_CFC_ (* Continuous Function Chart, elements in execution order *)
(* 60s *)
#0 AND(#2.Xm, SHU6_P2_UST_RE_RABOTA)
#1 ADD(SHU6_P2_M_MINSPEED, 0.1)
#2 LT_HZm20:ISTOK_LT(dost: TRUE, x: SHU6_P2_SPEEDMOTOR, ust: #1, shkal: -, gist: 1)
#3 INT_TO_TIME(SHU6_P2_M_ZAD_HZM20)
#4 MUL(#3, 1000)
#5 TON_HZm20:TON(IN: #0, PT: #4)
#6 AND(#5.Q, NOT SHU6_P2_M_SB2_STER_REG)
#7 SR_HZ20S60:SR(SET1: #6, RESET: SHU6_P2_SB)
#8 SHU6_P2_HZ20S60 <= #7.Q1
_END_CFC_
(* the same logic as Structured Text *)
(* 60s *)
_t19 := LT_HZm20.Xm AND SHU6_P2_UST_RE_RABOTA;
LT_HZm20(dost := TRUE, x := SHU6_P2_SPEEDMOTOR, ust := SHU6_P2_M_MINSPEED + 0.1, gist := 1);
TON_HZm20(IN := _t19, PT := INT_TO_TIME(SHU6_P2_M_ZAD_HZM20) * 1000);
SR_HZ20S60(SET1 := TON_HZm20.Q AND NOT SHU6_P2_M_SB2_STER_REG, RESET := SHU6_P2_SB);
SHU6_P2_HZ20S60 := SR_HZ20S60.Q1;
END_PROGRAM

(* POU TZBiS/TZB/Z_ALL, CFC *)
PROGRAM Z_ALL
VAR
	SR_Z_all: SR;
END_VAR
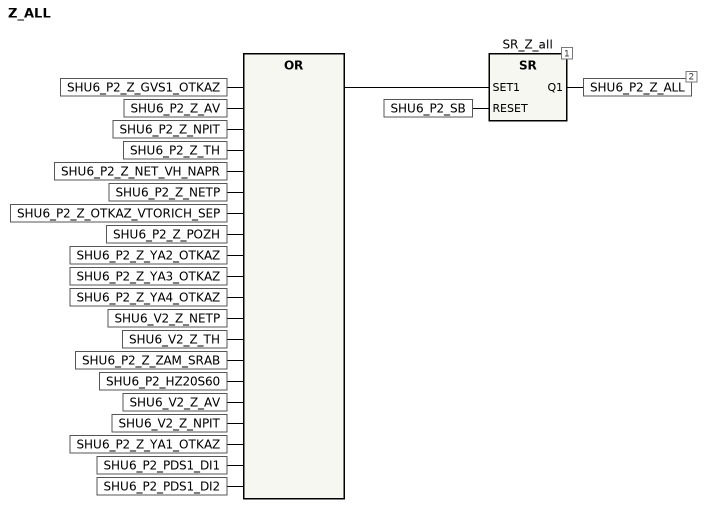
_CFC_ (* Continuous Function Chart, elements in execution order *)
#0 OR(SHU6_P2_Z_GVS1_OTKAZ, SHU6_P2_Z_AV, SHU6_P2_Z_NPIT, SHU6_P2_Z_TH, SHU6_P2_Z_NET_VH_NAPR, SHU6_P2_Z_NETP, SHU6_P2_Z_OTKAZ_VTORICH_SEP, SHU6_P2_Z_POZH, SHU6_P2_Z_YA2_OTKAZ, SHU6_P2_Z_YA3_OTKAZ, SHU6_P2_Z_YA4_OTKAZ, SHU6_V2_Z_NETP, SHU6_V2_Z_TH, SHU6_P2_Z_ZAM_SRAB, SHU6_P2_HZ20S60, SHU6_V2_Z_AV, SHU6_V2_Z_NPIT, SHU6_P2_Z_YA1_OTKAZ, SHU6_P2_PDS1_DI1, SHU6_P2_PDS1_DI2)
#1 SR_Z_all:SR(SET1: #0, RESET: SHU6_P2_SB)
#2 SHU6_P2_Z_ALL <= #1.Q1
_END_CFC_
(* the same logic as Structured Text *)
SR_Z_all(SET1 := SHU6_P2_Z_GVS1_OTKAZ OR SHU6_P2_Z_AV OR SHU6_P2_Z_NPIT OR SHU6_P2_Z_TH OR SHU6_P2_Z_NET_VH_NAPR OR SHU6_P2_Z_NETP OR SHU6_P2_Z_OTKAZ_VTORICH_SEP OR SHU6_P2_Z_POZH OR SHU6_P2_Z_YA2_OTKAZ OR SHU6_P2_Z_YA3_OTKAZ OR SHU6_P2_Z_YA4_OTKAZ OR SHU6_V2_Z_NETP OR SHU6_V2_Z_TH OR SHU6_P2_Z_ZAM_SRAB OR SHU6_P2_HZ20S60 OR SHU6_V2_Z_AV OR SHU6_V2_Z_NPIT OR SHU6_P2_Z_YA1_OTKAZ OR SHU6_P2_PDS1_DI1 OR SHU6_P2_PDS1_DI2, RESET := SHU6_P2_SB);
SHU6_P2_Z_ALL := SR_Z_all.Q1;
END_PROGRAM

(* POU TZBiS/TZB/Z_YA2_Otk, CFC *)
PROGRAM Z_YA2_Otk
VAR
	SR_YA2_Otkaz: SR;
	TON_YA2_Otk: TON;
	TON_YA2_N_OTKR: TON;
	TON_YA2_N_ZAKR: TON;
	TON_YA2_ZKR: TON;
	TON_AVT: TON;

	a: BOOL;
	b: BOOL;
	c: BOOL;
	d: BOOL;
	e: BOOL;
END_VAR
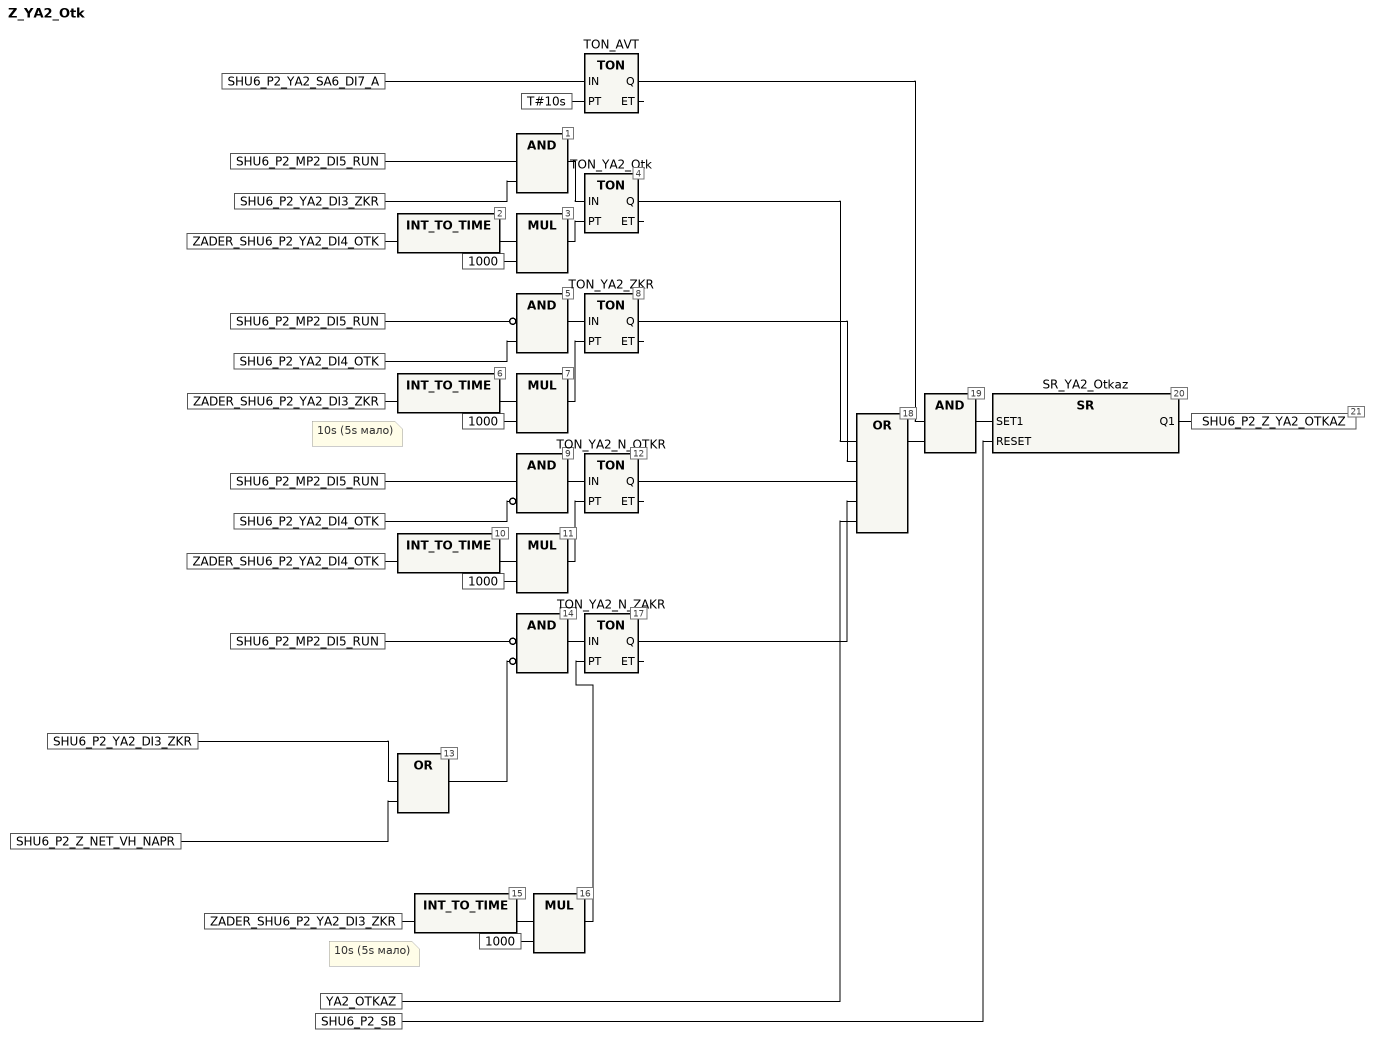
_CFC_ (* Continuous Function Chart, elements in execution order *)
(* 10s (5s мало) *)
(* 10s (5s мало) *)
#0 TON_AVT:TON(IN: SHU6_P2_YA2_SA6_DI7_A, PT: T#10s)
#1 AND(SHU6_P2_MP2_DI5_RUN, SHU6_P2_YA2_DI3_ZKR)
#2 INT_TO_TIME(ZADER_SHU6_P2_YA2_DI4_OTK)
#3 MUL(#2, 1000)
#4 TON_YA2_Otk:TON(IN: #1, PT: #3)
#5 AND(NOT SHU6_P2_MP2_DI5_RUN, SHU6_P2_YA2_DI4_OTK)
#6 INT_TO_TIME(ZADER_SHU6_P2_YA2_DI3_ZKR)
#7 MUL(#6, 1000)
#8 TON_YA2_ZKR:TON(IN: #5, PT: #7)
#9 AND(SHU6_P2_MP2_DI5_RUN, NOT SHU6_P2_YA2_DI4_OTK)
#10 INT_TO_TIME(ZADER_SHU6_P2_YA2_DI4_OTK)
#11 MUL(#10, 1000)
#12 TON_YA2_N_OTKR:TON(IN: #9, PT: #11)
#13 OR(SHU6_P2_YA2_DI3_ZKR, SHU6_P2_Z_NET_VH_NAPR)
#14 AND(NOT SHU6_P2_MP2_DI5_RUN, NOT #13)
#15 INT_TO_TIME(ZADER_SHU6_P2_YA2_DI3_ZKR)
#16 MUL(#15, 1000)
#17 TON_YA2_N_ZAKR:TON(IN: #14, PT: #16)
#18 OR(#4.Q, #8.Q, #12.Q, #17.Q, YA2_OTKAZ)
#19 AND(#0.Q, #18)
#20 SR_YA2_Otkaz:SR(SET1: #19, RESET: SHU6_P2_SB)
#21 SHU6_P2_Z_YA2_OTKAZ <= #20.Q1
_END_CFC_
(* the same logic as Structured Text *)
(* 10s (5s мало) *)
(* 10s (5s мало) *)
TON_AVT(IN := SHU6_P2_YA2_SA6_DI7_A, PT := T#10s);
TON_YA2_Otk(IN := SHU6_P2_MP2_DI5_RUN AND SHU6_P2_YA2_DI3_ZKR, PT := INT_TO_TIME(ZADER_SHU6_P2_YA2_DI4_OTK) * 1000);
TON_YA2_ZKR(IN := NOT SHU6_P2_MP2_DI5_RUN AND SHU6_P2_YA2_DI4_OTK, PT := INT_TO_TIME(ZADER_SHU6_P2_YA2_DI3_ZKR) * 1000);
TON_YA2_N_OTKR(IN := SHU6_P2_MP2_DI5_RUN AND NOT SHU6_P2_YA2_DI4_OTK, PT := INT_TO_TIME(ZADER_SHU6_P2_YA2_DI4_OTK) * 1000);
TON_YA2_N_ZAKR(IN := NOT SHU6_P2_MP2_DI5_RUN AND NOT (SHU6_P2_YA2_DI3_ZKR OR SHU6_P2_Z_NET_VH_NAPR), PT := INT_TO_TIME(ZADER_SHU6_P2_YA2_DI3_ZKR) * 1000);
SR_YA2_Otkaz(SET1 := TON_AVT.Q AND (TON_YA2_Otk.Q OR TON_YA2_ZKR.Q OR TON_YA2_N_OTKR.Q OR TON_YA2_N_ZAKR.Q OR YA2_OTKAZ), RESET := SHU6_P2_SB);
SHU6_P2_Z_YA2_OTKAZ := SR_YA2_Otkaz.Q1;
END_PROGRAM

(* POU TZBiS/TZB/Z_YA1_YA2_NPit, CFC *)
PROGRAM Z_YA1_YA2_NPit
VAR
	SR_YA1_YA2_NPit: SR;
	SR_IBP_NPit: SR;
	SR_A1_G1_NPit: SR;
	SR_A1_TV1_NPit: SR;
	SR_24V_NPit: SR;
END_VAR
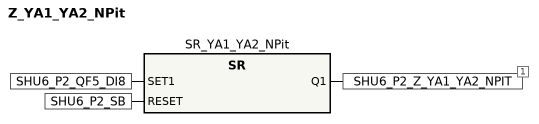
_CFC_ (* Continuous Function Chart, elements in execution order *)
#0 SR_YA1_YA2_NPit:SR(SET1: SHU6_P2_QF5_DI8, RESET: SHU6_P2_SB)
#1 SHU6_P2_Z_YA1_YA2_NPIT <= #0.Q1
_END_CFC_
(* the same logic as Structured Text *)
SR_YA1_YA2_NPit(SET1 := SHU6_P2_QF5_DI8, RESET := SHU6_P2_SB);
SHU6_P2_Z_YA1_YA2_NPIT := SR_YA1_YA2_NPit.Q1;
END_PROGRAM

(* POU TZBiS/TZB/Z_YA3_Otk, CFC *)
PROGRAM Z_YA3_Otk
VAR
	SR_YA3_Otk: SR;
	TON_YA3_Rassog: TON;
	RT_Rassog: R_TRIG;
	TON_YA3_Rassog1: TON;
	TIME_DELAY: TIME;
END_VAR
VAR (* helpers for the ST form of the networks *)
	_t14 : BOOL;
END_VAR
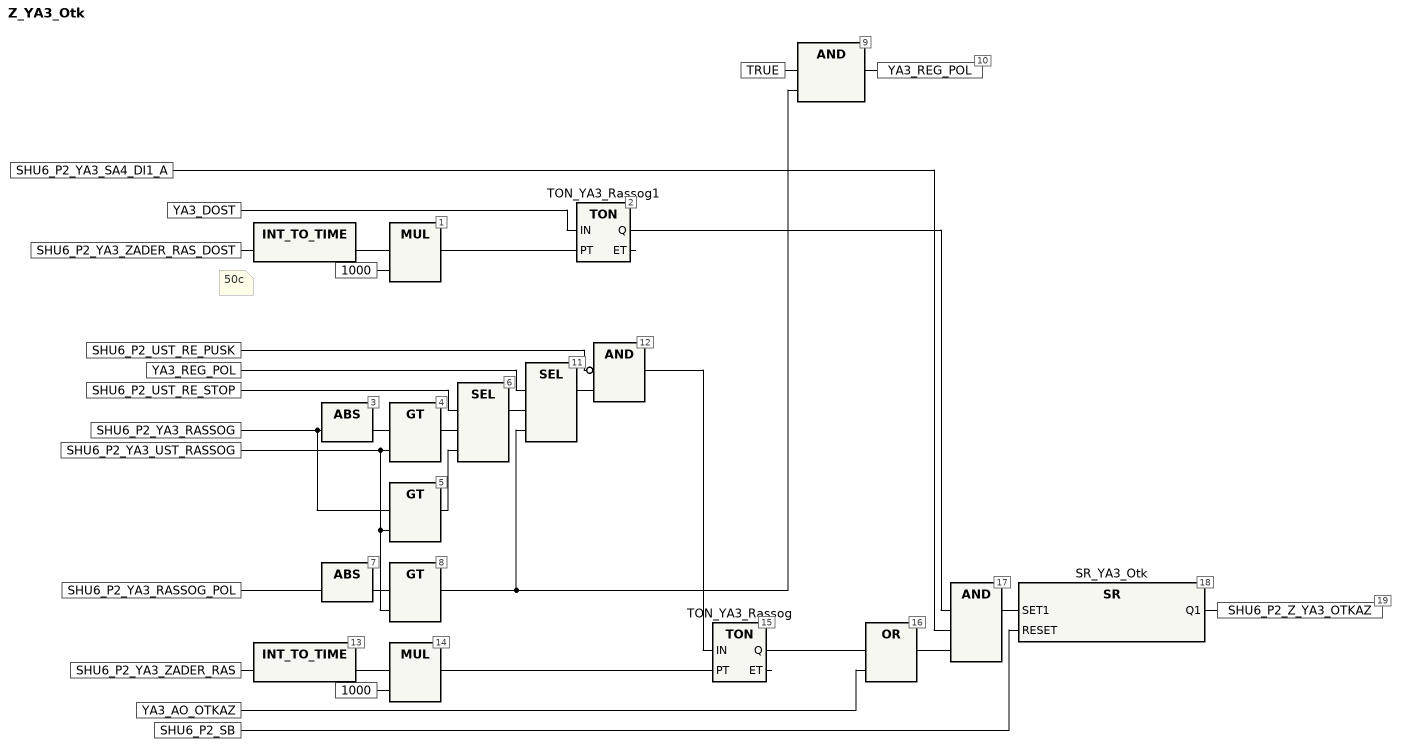
